{attribute 'GeneratedUsingTerminal: KL2652-0050'}
{attribute addProperty BoxType "KL2652-0050"}
{attribute addProperty Id "Channel_1AT %Q*Channel_6D8B740B0Channel_2AT %Q*Channel_6D8B740B0"}
{attribute addProperty CRC "334306021"}
{attribute addProperty Size "0"}
TYPE KL_13ED1AE5 :
STRUCT
	{attribute addProperty Name "Channel_1"}
	Channel_1 : Channel_6D8B740B;
	{attribute addProperty Name "Channel_2"}
	Channel_2 : Channel_6D8B740B;
END_STRUCT
END_TYPE

(* stored: Version 1.2.0.0, ProductVersion 3.1.4024.9
   DUT KL_13ED1AE5: Id {4bc8aff3-1f30-438f-8136-737a0b43f225} *)
